FUNCTION_BLOCK ConsoleHMI
  (* Standard: 61499-2 *)
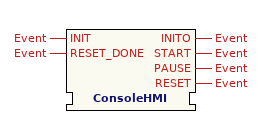
  EVENT_INPUT
    INIT;
    RESET_DONE;
  END_EVENT
  EVENT_OUTPUT
    INITO;
    START;
    PAUSE;
    RESET;
  END_EVENT
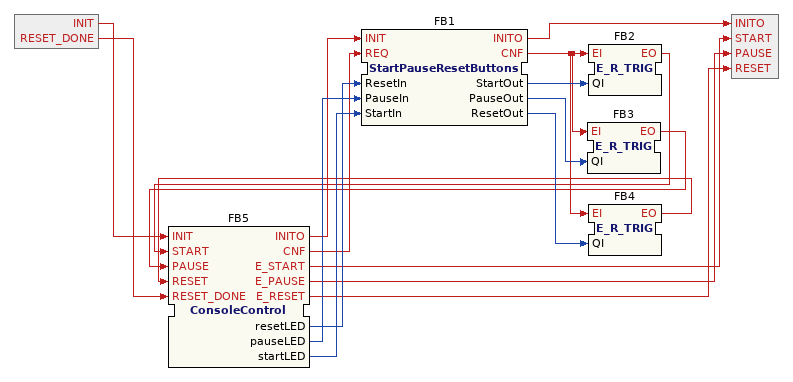
  FBS
    FB1 : StartPauseResetButtons;
    FB2 : E_R_TRIG;
    FB3 : E_R_TRIG;
    FB4 : E_R_TRIG;
    FB5 : ConsoleControl;
  END_FBS
  EVENT_CONNECTIONS
    INIT TO FB5.INIT;
    FB1.INITO TO INITO;
    FB1.CNF TO FB2.EI;
    FB1.CNF TO FB3.EI;
    FB1.CNF TO FB4.EI;
    FB5.INITO TO FB1.INIT;
    FB5.CNF TO FB1.REQ;
    FB2.EO TO FB5.START;
    FB3.EO TO FB5.PAUSE;
    FB4.EO TO FB5.RESET;
    RESET_DONE TO FB5.RESET_DONE;
    FB5.E_START TO START;
    FB5.E_PAUSE TO PAUSE;
    FB5.E_RESET TO RESET;
  END_CONNECTIONS
  DATA_CONNECTIONS
    FB1.StartOut TO FB2.QI;
    FB1.PauseOut TO FB3.QI;
    FB1.ResetOut TO FB4.QI;
    FB5.resetLED TO FB1.ResetIn;
    FB5.pauseLED TO FB1.PauseIn;
    FB5.startLED TO FB1.StartIn;
  END_CONNECTIONS
END_FUNCTION_BLOCK
